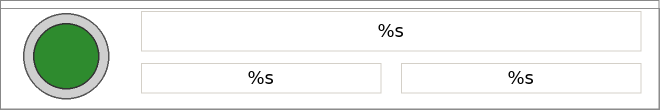
VISUALIZATION SingleDigitalInput  // 660x110
VAR_IN_OUT
	stDigitalInput : ST_VisuCtrlInputFrame;
END_VAR
    GroupBox (0,0 660x110)
        Lamp1 (16,6 100x100), variable: stDigitalInput.bIn, style: Lamp-Lamp1-Green
        Textfield (141,11 500x40), "%s", text variable: stDigitalInput.sName
        Textfield (141,63 240x30), "%s", text variable: stDigitalInput.sModuleType
        Textfield (401,63 240x30), "%s", text variable: stDigitalInput.sPortID
END_VISUALIZATION

(* stored: Version 1.1.0.1, ProductVersion 3.1.4024.12
   Visu SingleDigitalInput: Id {7c020ee1-48a4-4171-b4ce-2a0e57be811d} *)
